FUNCTION_BLOCK E_CTU (* Event driven up counter *)
  (* Standard: 61499-1 Annex 2; Description: Copyright (c) 2017 fortiss GmbH This program and the accompanying materials are made available under the terms of the Eclipse Public License 2.0 which is available at https://www.eclipse.org/legal/epl-2.0/ SPDX-License-Identifier: EPL-2.0 *)
  (* Version 1.0, 2017-09-21, Alois Zoitl, fortiss GmbH, initial API and implementation and/or initial documentation *)
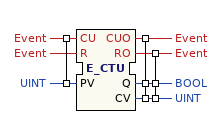
  EVENT_INPUT
    CU WITH PV; (* Count up *)
    R; (* Reset *)
  END_EVENT
  EVENT_OUTPUT
    CUO WITH Q, CV; (* Count up output *)
    RO WITH Q, CV; (* Reset output *)
  END_EVENT
  VAR_INPUT
    PV : UINT; (* Process Value *)
  END_VAR
  VAR_OUTPUT
    Q : BOOL; (* True if CV &gt;= PV *)
    CV : UINT; (* Counter Value *)
  END_VAR
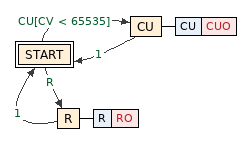
  EC_STATES
    START; (* Initial State *)
    CU : CU -> CUO;
    R : R -> RO;
  END_STATES
  EC_TRANSITIONS
    START TO CU := CU[CV < 65535];
    CU TO START := 1;
    START TO R := R;
    R TO START := 1;
  END_TRANSITIONS
  ALGORITHM R IN ST:
CV := 0;
Q := FALSE;
  END_ALGORITHM
  ALGORITHM CU IN ST:
CV := CV + 1;
Q  := (CV >= PV);
  END_ALGORITHM
  SERVICE left interface/right interface (* Event driven up counter *)
    SEQUENCE Service Sequence
      left interface.CU(CV:=0) -> left interface.CUO(CV:=1);
    END_SEQUENCE
    SEQUENCE Service Sequence {SET_ATTRIBUTE(StartState, START)}
      left interface.CU() -> left interface.CUO(Q:=BOOL#TRUE; CV:=UINT#1;);
      left interface.CU() -> left interface.CUO(Q:=BOOL#TRUE; CV:=UINT#2;);
    END_SEQUENCE
    SEQUENCE Service Sequence {SET_ATTRIBUTE(StartState, START)}
      left interface.CU() -> left interface.CUO(Q:=BOOL#TRUE; CV:=UINT#1;);
      left interface.CU() -> left interface.CUO(Q:=BOOL#TRUE; CV:=UINT#1;);
      left interface.CU() -> left interface.CUO(Q:=BOOL#TRUE; CV:=UINT#1;);
      left interface.CU() -> left interface.CUO(Q:=BOOL#TRUE; CV:=UINT#1;);
    END_SEQUENCE
  END_SERVICE
END_FUNCTION_BLOCK
